TYPE E_LinkState :
(
    eDisconnected   := 0,
    eConnecting     := 1,
    eConnected      := 2,
    eError          := 3,
    eReconnectWait  := 4
);
END_TYPE

(* stored: Version 1.1.0.1, ProductVersion 3.1.4026.18
   DUT E_LinkState: Id {1a969a5f-3642-46a1-a80a-498c7698b082} *)
